Yaskawa INFORM job: UNCLAMP_GRIPPER.JBI

/JOB
//NAME UNCLAMP_GRIPPER
//POS
///NPOS 0,0,0,0,0,0
//INST
///DATE 2018/08/30 13:35
///ATTR SC,RW
NOP
DOUT OT#(20) OFF
PULSE OT#(21)
IFTHEN B021=1
	 WAIT IN#(9)=ON
ENDIF
TIMER T=0.50
SET B011 0
SET B016 0
END
